(* CoDeSys 2.3.9.47 project: test.pro *)
(* Libraries: Iecsfc.lib 12.5.98 12:03:00, STANDARD.LIB 5.6.98 12:03:02 *)

(* Task configuration *)
TASK Standard (PRIORITY := 0, INTERVAL := T#1000ms);
	MAIN
END_TASK

(* Data type *)
TYPE pump_structures :
STRUCT
	x : POINTER TO INT;
	y: POINTER TO INT ;
END_STRUCT
END_TYPE

(* POU MAIN, ST *)
PROGRAM MAIN
VAR
	z : pump_structures;
	x : INT;
	y : INT;
END_VAR
TANK_STREAM1_A;


(*lets experiment with structure and pointers*)

z.x := ADR(x);

z.x^ := 10;

z.x^;
END_PROGRAM

(* POU TANK_STREAM1_A, SFC *)
PROGRAM TANK_STREAM1_A
VAR
	Trans4: BOOL;
	Trans3: BOOL;
	Trans2: BOOL;
	Trans1: BOOL;
END_VAR
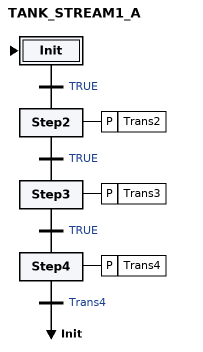
INITIAL_STEP Init:
END_STEP
TRANSITION FROM Init TO Step2 := TRUE;
END_TRANSITION
STEP Step2:
	Trans2(P);
END_STEP
TRANSITION FROM Step2 TO Step3 := TRUE;
END_TRANSITION
STEP Step3:
	Trans3(P);
END_STEP
TRANSITION FROM Step3 TO Step4 := TRUE;
END_TRANSITION
STEP Step4:
	Trans4(P);
END_STEP
TRANSITION FROM Step4 TO Init := Trans4;
END_TRANSITION
END_PROGRAM

(* POU testing, ST *)
FUNCTION_BLOCK testing
VAR_INPUT
END_VAR
VAR_OUTPUT
END_VAR
VAR
END_VAR
VAR_IN_OUT
	z:pump_structures;
END_VAR
z.x^ := z.x^ + 1;
END_FUNCTION_BLOCK
